// TIA Portal V20 export
DATA_BLOCK "ControlNodes"   // DB136
// stored: MemoryReserve 100, Namespace Unit1.Em13
   VAR
      em : "LAF_typeEmControlNode";
      emstate { S7_SetPoint := 'True'} : "LUC_typeStates";
      cm : "Unit1.Em13.typeCmControlNode";
      citiMap : Struct
         PMC : "LER_PMC_Input_Data";
         FlexNet { S7_SetPoint := 'True'} : "LER_FlexNet_Data";
      END_STRUCT;
      jrUnloadingPnP : "Unit1.Em13.typeSequenceControlNode";
      emData : "LER_typePartData";
      unitCommunication : "Unit1.Em13.typeUnitCommunicationControlNode";
      FATMode : "LER_TypeFATMode_ModeSelect";
      SpecialFunctionMode : Struct
         DryRun : Struct
            JRdetectPV : Array[0..15] of Bool;
         END_STRUCT;
      END_STRUCT;
      cmJRUnloadingPnPSafetyPin : "LBC_typeDigitalSignalControlNode";
      cmJRUnloadingPnPJRDetect : "LBC_typeDigitalSignalControlNode";
      cmJRUnloadingPnPAxisX : "LBC_typeAxis64PosControlNode";
      cmJRUnloadingPnPAxisZ : "LBC_typeAxis64PosControlNode";
      cmJRUnloadingPnPAxisC : "LBC_typeAxis64PosControlNode";
      cmJRUnloadingPnPClampOpenClose : "LBC_typeTwoWayActuatorControlNode";
      ConVisionComplete { S7_SetPoint := 'True'} : Bool;   // Vision complete Memory
   END_VAR
BEGIN
END_DATA_BLOCK
